(* IEC 61131-3 sources: CS_4_Aufzugsteuerung/src/Stations/CP112/Steuerung/Class/clsTimer, 1 file *)

(* ---- clsTimer.st ---- *)
(*!
<Class
	Name               = "clsTimer"
	Revision           = "0.0"
	RealtimeTask       = "false"
	CyclicTask         = "true"
	DefCyclictime      = "50 ms"
	BackgroundTask     = "false"
	Sigmatek           = "false"
	OSInterface        = "false"
	HighPriority       = "false"
	Automatic          = "false"
	UpdateMode         = "Prescan"
	SharedCommandTable = "true"
	Objectsize         = "(300,120)">
	<Channels>
		<Server Name="ClassSvr" Visualized="false" Initialize="false" WriteProtected="true" Retentive="false"/>
	</Channels>
</Class>
*)
clsTimer : CLASS
  //Servers:
	ClassSvr 	: SvrChCmd_DINT;
  //Clients:
  //Variables:
		vTime 	: UDINT;
		vTimeOffset 	: UDINT;
		vIsRunning 	: BOOL;
		vlsElapsed 	: DINT;
  //Functions:

	FUNCTION VIRTUAL GLOBAL CyWork
		VAR_INPUT
			EAX 	: UDINT;
		END_VAR
		VAR_OUTPUT
			state (EAX) 	: UDINT;
		END_VAR;

	FUNCTION VIRTUAL GLOBAL RtWork
		VAR_INPUT
			EAX 	: UDINT;
		END_VAR
		VAR_OUTPUT
			state (EAX) 	: UDINT;
		END_VAR;

	FUNCTION GLOBAL start
		VAR_INPUT
			_time 	: UDINT;
		END_VAR;

	FUNCTION GLOBAL reset;

	FUNCTION GLOBAL elapsed
		VAR_OUTPUT
			isElapsed 	: BOOL;
		END_VAR;

	FUNCTION GLOBAL running
		VAR_OUTPUT
			isRunning 	: BOOL;
		END_VAR;

	FUNCTION GLOBAL remaining
		VAR_OUTPUT
			remaining 	: UDINT;
		END_VAR;
  //Tables:
	FUNCTION @STD
		VAR_OUTPUT
			ret_code	: CONFSTATES;
		END_VAR;
	FUNCTION GLOBAL TAB @CT_;
END_CLASS;

FUNCTION GLOBAL clsTimer::start
	VAR_INPUT
		_time 	: UDINT;
	END_VAR

  // Merken des Offsets
  vTimeOffset := _time;

  //Merken der Startzeit
  vTime := ops.tAbsolute;

  vIsRunning := TRUE;

END_FUNCTION

FUNCTION GLOBAL clsTimer::reset

  vTimeOffset := 0;
  vTime := 0;
  vIsRunning := FALSE;

END_FUNCTION

FUNCTION GLOBAL clsTimer::elapsed
	VAR_OUTPUT
		isElapsed 	: BOOL;
	END_VAR

  IF vIsRunning AND ((ops.tAbsolute - vTime) >= vTimeOffset) THEN
    isElapsed := TRUE;
    vIsRunning := FALSE;
  ELSE
    isElapsed := FALSE;
  END_IF;

  vlsElapsed := isElapsed;

END_FUNCTION

FUNCTION GLOBAL clsTimer::running
	VAR_OUTPUT
		isRunning 	: BOOL;
	END_VAR

  IF vIsRunning THEN
    isRunning := TRUE;
  ELSE
    isRunning := FALSE;
  END_IF;

END_FUNCTION

FUNCTION GLOBAL clsTimer::remaining
	VAR_OUTPUT
		remaining 	: UDINT;
	END_VAR

  IF NOT vIsRunning THEN
      remaining := 0;
  ELSIF (ops.tAbsolute - vTime) >= vTimeOffset THEN
      remaining := 0;
  ELSE
      remaining := vTimeOffset - (ops.tAbsolute - vTime);
  END_IF;

END_FUNCTION

FUNCTION VIRTUAL GLOBAL clsTimer::RtWork
	VAR_INPUT
		EAX 	: UDINT;
	END_VAR
	VAR_OUTPUT
		state (EAX) 	: UDINT;
	END_VAR

	state := READY;

END_FUNCTION

FUNCTION VIRTUAL GLOBAL clsTimer::CyWork
	VAR_INPUT
		EAX 	: UDINT;
	END_VAR
	VAR_OUTPUT
		state (EAX) 	: UDINT;
	END_VAR

	state := READY;

END_FUNCTION
